SUBAPPLICATION Sample (* Subapplication Type *)
  (* Standard: 61499-2 *)
  (* Version 1.0, 2023-02-17, Franz *)
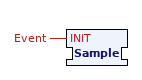
  EVENT_INPUT
    INIT;
  END_EVENT
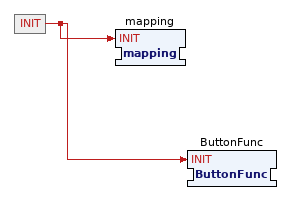
  SUBAPPS
    mapping : mapping;
    ButtonFunc : ButtonFunc;
  END_SUBAPPS
  EVENT_CONNECTIONS
    INIT TO mapping.INIT;
    INIT TO ButtonFunc.INIT;
  END_CONNECTIONS
END_SUBAPPLICATION
